{attribute 'GeneratedUsingTerminal: EL7031-0030-0016'}
{attribute addProperty BoxType "EL7031-0030-0016"}
{attribute addProperty Id "AdsAddrAT %I*.TcoAmsAddr0Chn0AT %I*USINT1Chn1AT %I*USINT1Chn2AT %I*USINT1Chn3AT %I*USINT1StateAT %I*UINT2"}
{attribute addProperty CRC "4153865593"}
{attribute addProperty Size "6"}
TYPE InfoData_F796F579 :
STRUCT
	{attribute addProperty Name "AdsAddr"}
	AdsAddr AT %I* : .TcoAmsAddr;
	{attribute addProperty Name "Chn0"}
	Chn0 AT %I* : USINT;
	{attribute addProperty Name "Chn1"}
	Chn1 AT %I* : USINT;
	{attribute addProperty Name "Chn2"}
	Chn2 AT %I* : USINT;
	{attribute addProperty Name "Chn3"}
	Chn3 AT %I* : USINT;
	{attribute addProperty Name "State"}
	State AT %I* : UINT;
END_STRUCT
END_TYPE

(* stored: Version 1.2.0.0, ProductVersion 3.1.4024.9
   DUT InfoData_F796F579: Id {ea26d16c-b6d9-4355-84f1-6e72785c3153} *)
